Fanuc KAREL source: kt00157.KL

-- PROVISIONAL review KL for V1013-1; original PC SHA256 cfd7921de0c1f5f1cbcd4f2adfdeab092697b49484044a29387deea84f9cf4e1
-- Incomplete behavior may be omitted. Consult companion uncertainty JSON. Do not deploy.
PROGRAM KT00157
%NOLOCKGROUP
VAR
  OUT : INTEGER
-- UNRESOLVED_DECL H1 type=002017
-- UNRESOLVED_DECL Y2 type=002018
BEGIN
  -- UNRESOLVED_PC offsets 5-19; opcodes 2E,22,9D,33,B4
  -- UNRESOLVED_PC offsets 24-38; opcodes 2E,22,9D,33,B2
  -- UNRESOLVED_PC offsets 43-68; opcodes 22,9D,33,B3,22,9D,33,B1,55,23
  -- UNRESOLVED_PC offsets 73-77; opcodes 7F
END KT00157
